FUNCTION FN_ResolveDBStatusRouteDevice : cResolvedDBStatusRoute

VAR_IN_OUT
	Device: DeviceData;
END_VAR

VAR_INPUT
	RouteToWork: STRING(30);
END_VAR

VAR
	tempResolved: cResolvedDBStatusRoute;
END_VAR


//Deafault to none in case logic fails
tempResolved := cResolvedDBStatusRoute.None;

// Check satus indicates unknown device	
IF Device.Status = cDBDeviceStatus.Unknown THEN
	tempResolved := cResolvedDBStatusRoute.UnknownDevice;
// Deal with normal status devices
ELSIF Device.Status = cDBDeviceStatus.Normal THEN
	IF Device.Route = cDBDetailRoute.PuckException THEN
		tempResolved := cResolvedDBStatusRoute.Normal_RoutedException;
	ELSIF Device.Route = cDBDetailRoute.Consolidation THEN
		tempResolved := cResolvedDBStatusRoute.Normal_RoutedConsolidation;
	ELSIF Device.Route = RouteToWork AND RouteToWork <> '' THEN
		tempResolved := cResolvedDBStatusRoute.Normal_RoutedThisStation;
	ELSE
		tempResolved := cResolvedDBStatusRoute.Normal_RoutedOtherStation;
	END_IF
// Only thing left is non-normal devices which go to exception by default.
ELSE
	tempResolved := cResolvedDBStatusRoute.NonNormal_RoutedException;
END_IF
	
FN_ResolveDBStatusRouteDevice := tempResolved;

END_FUNCTION

(* stored: Version 1.1.0.1, ProductVersion 3.1.4024.6
   POU FN_ResolveDBStatusRouteDevice: Id {b6fd4710-bb30-40f2-8da3-579298a72e24}, SpecialFunc None *)
